// TIA Portal V21 export
FUNCTION_BLOCK "RoutingParts"   // FB42, LAD
   VAR_TEMP   // added for the SCL form of the ladder/FBD networks
      _variant1 : Variant;
   END_VAR
BEGIN

REGION Network 1: Nested OR branches
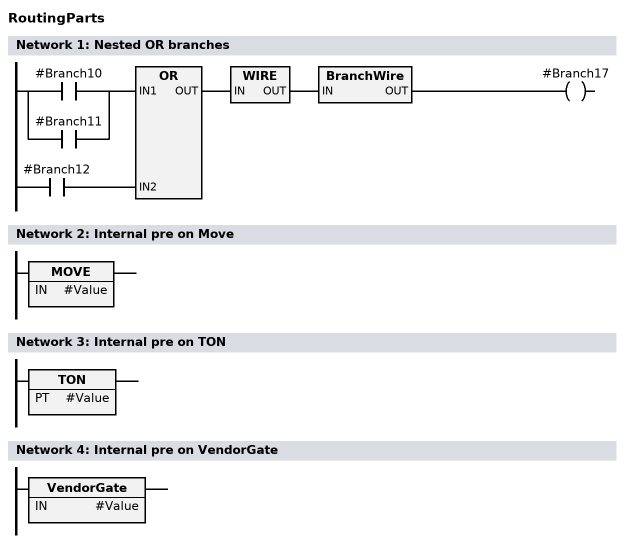
   // no SCL statement known for BranchWire, Wire: written as a call
   #_variant1 := (#Branch10 OR #Branch11) OR #Branch12;
   #Branch17 := BranchWire(Wire(#_variant1));
END_REGION

REGION Network 2: Internal pre on Move
   // no SCL statement known for Move: written as a call
END_REGION

REGION Network 3: Internal pre on TON
   // no SCL statement known for TON: written as a call
END_REGION

REGION Network 4: Internal pre on VendorGate
   // no SCL statement known for VendorGate: written as a call
END_REGION
END_FUNCTION_BLOCK
